FUNCTION_BLOCK FB_Axis EXTENDS FB_Base IMPLEMENTS I_Axis
VAR_INPUT
END_VAR
VAR_OUTPUT
END_VAR
VAR
END_VAR

METHOD InPosition : BOOL
VAR_INPUT
END_VAR
END_METHOD

METHOD MoveAbsolute : BOOL
VAR_INPUT
	target : REAL;
END_VAR
Tc2_System.ADSLOGSTR(0, CONCAT('axis move to position ', TO_STRING(target)), '');
END_METHOD

END_FUNCTION_BLOCK

(* stored: Version 1.1.0.1
   POU FB_Axis: Id {24a9cdac-e68f-40e5-8ce6-e0b3ae83894a}, SpecialFunc None
   Method InPosition: Id {031a12bb-7b5c-4e2e-a15a-8d27a2e89b04}
   Method MoveAbsolute: Id {1175759c-5dea-4004-a9bd-113763a78787} *)
